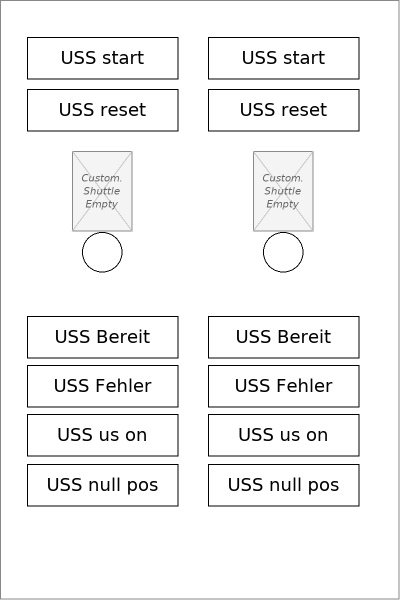
VISUALIZATION VISU_ST150  // 400x600
    RoundedRectangle (27,316 151x42), "USS Bereit", colour toggle: GVL.st150_aut.fb_Uss.xIN_welding_bits.Bereit
    RoundedRectangle (27,365 151x42), "USS Fehler", colour toggle: GVL.st150_aut.fb_Uss.xIN_welding_bits.Fehler
    RoundedRectangle (27,414 151x42), "USS us on", colour toggle: GVL.st150_aut.fb_Uss.xIN_welding_bits.US_on
    RoundedRectangle (27,464 151x42), "USS null pos", colour toggle: GVL.st150_aut.fb_Uss.xIN_welding_bits.NullPosition
    RoundedRectangle (27,37 151x42), "USS start", colour toggle: GVL.st150_aut.fb_Uss.xOUT_welding_bits.Start
    RoundedRectangle (27,89 151x42), "USS reset", colour toggle: GVL.st150_aut.fb_Uss.xOUT_welding_bits.Reset
    Ellipse (82,232 40x40), colour toggle: GVL.st150_aut.fb_Uss.xIN_capDetector
    Image (72,151 60x80), angle 90, invisible if: NOT __ISVALIDREF(GVL.st150_aut._Mover), image: Custom.Shuttle Empty
    RoundedRectangle (208,316 151x42), "USS Bereit", colour toggle: GVL.st155_aut.fb_Uss.xIN_welding_bits.Bereit
    RoundedRectangle (208,365 151x42), "USS Fehler", colour toggle: GVL.st155_aut.fb_Uss.xIN_welding_bits.Fehler
    RoundedRectangle (208,414 151x42), "USS us on", colour toggle: GVL.st155_aut.fb_Uss.xIN_welding_bits.US_on
    RoundedRectangle (208,464 151x42), "USS null pos", colour toggle: GVL.st155_aut.fb_Uss.xIN_welding_bits.NullPosition
    RoundedRectangle (208,37 151x42), "USS start", colour toggle: GVL.st155_aut.fb_Uss.xOUT_welding_bits.Start
    RoundedRectangle (208,89 151x42), "USS reset", colour toggle: GVL.st155_aut.fb_Uss.xOUT_welding_bits.Reset
    Ellipse (263,232 40x40), colour toggle: GVL.st155_aut.fb_Uss.xIN_capDetector
    Image (253,151 60x80), angle 90, invisible if: NOT __ISVALIDREF(GVL.st155_aut._Mover), image: Custom.Shuttle Empty
END_VISUALIZATION

(* stored: Version 1.1.0.1, ProductVersion 3.1.4024.6
   Visu VISU_ST150: Id {e3b53aa0-20d2-457e-acb8-c72d6d9848ef} *)
